INTERFACE I_LinearContinuousDrive EXTENDS I_LinearDrive, I_ContinuousDrive

END_INTERFACE

(* stored: Version 1.1.0.1, ProductVersion 3.1.4024.11
   Itf I_LinearContinuousDrive: Id {258447d5-36e1-40d4-8298-a7421bbca512} *)
